// TIA Portal V21 export
DATA_BLOCK "数据块_1"   // DB2
{ S7_Optimized_Access := 'TRUE' }
// stored: MemoryReserve 100
   VAR
      Timer1 : TON_TIME;
      Timer2 { S7_SetPoint := 'True'} : TON_TIME;
      当前扭矩浮点数 { S7_SetPoint := 'True'} : Real;
      正向扭矩设定 { S7_SetPoint := 'True'} : Real;
      负向扭矩设定 { S7_SetPoint := 'True'} : Real;
   END_VAR
BEGIN
END_DATA_BLOCK
